ABB RobotStudio station: IRB120-Estacion.rsstn

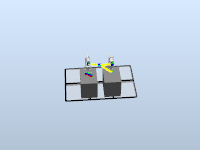
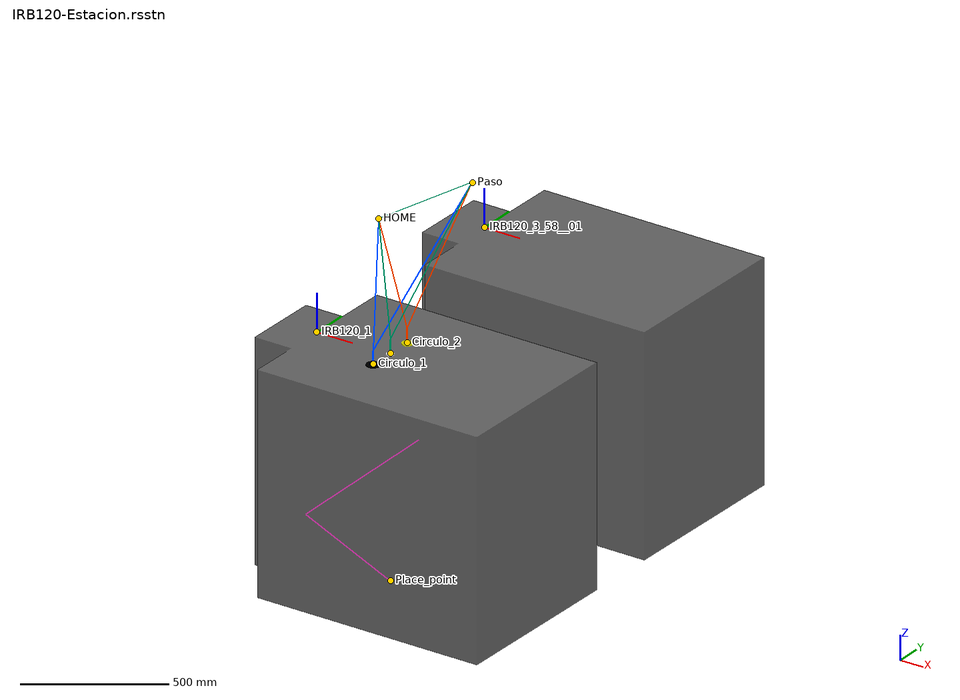
[picture v1: parts stored in the station drawn from their meshes, with robot base, taught points and paths (robot models come from the ABB library and are not in the file)]
Station IRB120 (saved by RobotStudio 21.4.9700.0)
Controller Controlador3, task T_ROB1: task frame (RAPID world) sits at (0, 980, 850) mm in the station
Controller Controlador1, task T_ROB1: task frame (RAPID world) sits at (0, 0, 850) mm in the station
Controller Controlador1
  mechanical unit ROB_1: IRB120_1, 6 joints, base frame (0, 0, 0) mm
Controller Controlador3
  mechanical unit ROB_1: IRB120_3_58__01, 6 joints, base frame (0, 0, 0) mm
Layout (positions relative to the parent item):
  - Base_2 [part] at (-150, 830, 0) mm, size 300 x 300 x 850 mm
  - IRB120_1 [mechanism, from Robots\IRB120_3_58_G_01.rslib] at (0, 0, 850) mm; joint values [0.0979, -0.2482, 0.2787, 0.0002, 1.5414, 0.0978] (rad or m)
  - Base_1 [part] at (-150, -150, 0) mm, size 300 x 300 x 850 mm
  - Ventosa_1 [mechanism, from Libraries\Ventosa.rslib] at (236.44, 23.25, 1390.49) mm, rotated rx 180 ry -0.06 rz -179.99 deg
  - Ventosa_2 [mechanism, from Libraries\Ventosa.rslib] at (364.35, 980, 1444) mm, rotated rx 180 ry 60 rz 180 deg
  - Mesa_1 [part], size 900 x 700 x 850 mm
  - Mesa_2 [part], size 900 x 700 x 850 mm
  - Circulo1 [part] at (300, 0, 850) mm, rotated rx 180 ry 0 rz 180 deg, size 30 x 29.8 x 5 mm
  - Circulo2 [part] at (300, 100, 850) mm, rotated rx 180 ry 0 rz 180 deg, size 40 x 39.8 x 5 mm
  - Circulo3 [part] at (300, -100, 850) mm, rotated rx 180 ry 0 rz 180 deg, size 50 x 49.7 x 5 mm
  - IRB120_3_58__01 [mechanism, from Robots\IRB120_3_58_G_01.rslib] at (0, 980, 850) mm; joint values [0, 0, 0, 0, 0.5236, 0] (rad or m)
Attachment: Ventosa_1 is attached to IRB120_1 / Link6
Attachment: Ventosa_2 is attached to IRB120_3_58__01 / Link6
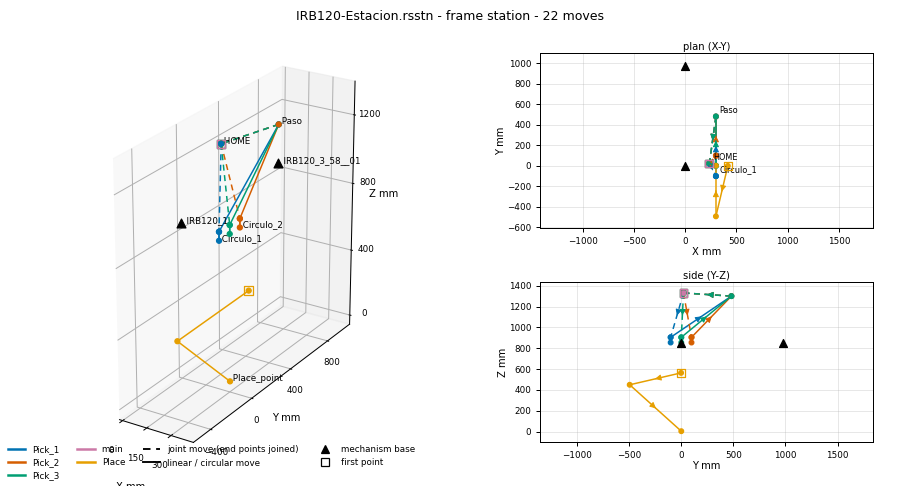
[picture p0: tool path of IRB120-Estacion.rsstn in frame station, 22 of 32 moves have a stored position in this frame; points joined in program order, loops and branches not executed]
Targets, tools, work objects and paths stored in the station, written as RAPID:
! task (no controller)
MODULE ROB1_Sim
  CONST robtarget Prueba:=[[0,0,5],[0,0,1,0],[0,0,0,0],[9E+09,9E+09,9E+09,9E+09,9E+09,9E+09]];
ENDMODULE

! task T_ROB1
MODULE ROB1_Sim
  PERS tooldata Ventosa:=[TRUE,[[0,0,60],[1,0,0,0]],[0.4,[0,0,1],[1,0,0,0],0,0,0]];
  CONST robtarget HOME:=[[236.38,23.25,480.49],[0.000528585,0.000071894,-1,-0.000034913],[0,0,0,0],[9E+09,9E+09,9E+09,9E+09,9E+09,9E+09]];
  CONST robtarget Circulo_1:=[[300,-100,5],[0,0,1,0],[-1,0,-1,0],[9E+09,9E+09,9E+09,9E+09,9E+09,9E+09]];
  CONST robtarget Circulo_2:=[[300,100,5],[0,0,1,0],[0,0,0,0],[9E+09,9E+09,9E+09,9E+09,9E+09,9E+09]];
  CONST robtarget Circulo_3:=[[300,2,5],[0,0,1,0],[0,0,0,0],[9E+09,9E+09,9E+09,9E+09,9E+09,9E+09]];
  CONST robtarget Paso:=[[300,482.5,450],[0.5,-0.5,0.5,0.5],[0,1,-1,0],[9E+09,9E+09,9E+09,9E+09,9E+09,9E+09]];
  CONST robtarget Prueba_10:=[[300,0,5],[0,0,1,0],[0,0,0,0],[9E+09,9E+09,9E+09,9E+09,9E+09,9E+09]];
  PROC Pick_1()
    MoveJ HOME,v100,fine,Ventosa\WObj:=wobj0;
    MoveJ Offs(Circulo_1,0,0,50),v100,fine,Ventosa\WObj:=wobj0;
    MoveL Circulo_1,v10,fine,Ventosa\WObj:=wobj0;
    MoveJ Offs(Circulo_1,0,0,50),v10,fine,Ventosa\WObj:=wobj0;
    MoveL Paso,v100,fine,Ventosa\WObj:=wobj0;
    MoveJ HOME,v100,fine,Ventosa\WObj:=wobj0;
  ENDPROC
  PROC Pick_2()
    MoveJ HOME,v100,fine,Ventosa\WObj:=wobj0;
    MoveJ Offs(Circulo_2,0,0,50),v100,fine,Ventosa\WObj:=wobj0;
    MoveL Circulo_2,v10,fine,Ventosa\WObj:=wobj0;
    MoveJ Offs(Circulo_2,0,0,50),v10,fine,Ventosa\WObj:=wobj0;
    MoveL Paso,v100,fine,Ventosa\WObj:=wobj0;
    MoveJ HOME,v100,fine,Ventosa\WObj:=wobj0;
  ENDPROC
  PROC Pick_3()
    MoveJ HOME,v100,fine,Ventosa\WObj:=wobj0;
    MoveJ Offs(Circulo_3,0,0,50),v100,fine,Ventosa\WObj:=wobj0;
    MoveL Circulo_3,v10,fine,Ventosa\WObj:=wobj0;
    MoveJ Offs(Circulo_3,0,0,50),v10,fine,Ventosa\WObj:=wobj0;
    MoveL Paso,v100,fine,Ventosa\WObj:=wobj0;
    MoveJ HOME,v100,fine,Ventosa\WObj:=wobj0;
  ENDPROC
ENDMODULE

! task T_ROB1
MODULE ROB1_Hanoi
  PROC main()
    MoveJ HOME,fast_speed,fine,vacuum_tool\WObj:=wobj0;
    TCP_connect;
    get_initial_state;
    TCP_close;
  ENDPROC
  PROC TCP_connect()
  ENDPROC
  PROC TCP_close()
  ENDPROC
  PROC get_initial_state()
    get_number_of_pieces;
  ENDPROC
  PROC get_number_of_pieces()
  ENDPROC
ENDMODULE

! task T_ROB1
MODULE Data
  PERS tooldata vacuum_tool:=[TRUE,[[0,0,60],[1,0,0,0]],[0.4,[0,0,1],[1,0,0,0],0,0,0]];
  TASK PERS wobjdata wo_b:=[FALSE,TRUE,"",[[448.203,36.8258,60.9458],[0.999999,-0.000331686,0.000243147,0.00150912]],[[56.8092,77.6912,0],[1,0,0,0]]];
  TASK PERS wobjdata wo_a:=[FALSE,TRUE,"",[[448.203,36.8258,60.9458],[0.999999,-0.000331686,0.000243147,0.00150912]],[[-56.0707,-122.147,0],[1,0,0,0]]];
ENDMODULE

! task T_ROB1
MODULE Hanoi_solver
  PROC initialize_desired_state()
  ENDPROC
ENDMODULE

! task T_ROB1
MODULE Module1
  PROC main()
  ENDPROC
ENDMODULE

! task T_ROB1
MODULE ROB2_Sim
  CONST robtarget HOME:=[[416.3153533,0,564],[0.5,0,0.866025404,0],[0,0,0,0],[9E+09,9E+09,9E+09,9E+09,9E+09,9E+09]];
  CONST robtarget Paso:=[[300,-492.5,450],[0.5,0.5,0.5,-0.5],[-1,-2,1,0],[9E+09,9E+09,9E+09,9E+09,9E+09,9E+09]];
  CONST robtarget Place_point:=[[300,2,5],[0,0,1,0],[0,0,0,0],[9E+09,9E+09,9E+09,9E+09,9E+09,9E+09]];
  PERS tooldata Ventosa:=[TRUE,[[0,0,60],[1,0,0,0]],[0.4,[0,0,1],[1,0,0,0],0,0,0]];
  PROC Place()
    MoveL HOME,v1000,z100,Ventosa\WObj:=wobj0;
    MoveL Paso,v1000,z100,Ventosa\WObj:=wobj0;
    MoveL Place_point,v1000,z100,Ventosa\WObj:=wobj0;
  ENDPROC
ENDMODULE

! task T_ROB1
MODULE ROB2_Hanoi
  PROC main()
    MoveJ \WObj:=wobj0;
    TCP_connect;
  ENDPROC
  PROC TCP_connect()
  ENDPROC
  PROC TCP_close()
  ENDPROC
  PROC get_initial_state()
  ENDPROC
  PROC place_on_C()
    MoveJ Offs(passing_point,0,50,0)\WObj:=wobj0;
    MoveL \WObj:=wobj0;
    WaitTime 0.5;
    MoveL Offs(passing_point,0,50,0)\WObj:=wobj0;
    MoveJ \WObj:=wobj0;
    MoveJ Offs(placing_point,0,0,(piece_height*pieces_on_C)+50);
    MoveL Offs(placing_point,0,0,(piece_height*pieces_on_C));
    WaitTime 0.5;
    MoveL Offs(placing_point,0,0,(piece_height*pieces_on_C)+50);
    MoveJ \WObj:=wobj0;
  ENDPROC
  PROC pick_and_pass()
    MoveJ Offs(placing_point,0,0,(piece_height*pieces_on_C)+50);
    MoveL Offs(placing_point,0,0,(piece_height*pieces_on_C));
    WaitTime 0.5;
    MoveL Offs(placing_point,0,0,(piece_height*pieces_on_C)+50);
    MoveJ \WObj:=wobj0;
    MoveJ Offs(passing_point,0,50,0)\WObj:=wobj0;
    MoveL \WObj:=wobj0;
    WaitTime 0.5;
    WaitTime 0.5;
    MoveL Offs(passing_point,0,50,0)\WObj:=wobj0;
    MoveJ \WObj:=wobj0;
  ENDPROC
ENDMODULE

! task T_ROB1
MODULE Module1
  CONST robtarget Target_10:=[[416.3153533,0,564],[0.5,0,0.866025404,0],[0,0,0,0],[9E+09,9E+09,9E+09,9E+09,9E+09,9E+09]];
ENDMODULE

! task T_ROB1
MODULE Data
  PERS tooldata vacuum:=[TRUE,[[0,0,0],[1,0,0,0]],[1,[0,0,0.001],[1,0,0,0],0,0,0]];
  TASK PERS wobjdata wo_c:=[FALSE,TRUE,"",[[0,0,0],[1,0,0,0]],[[0,0,0],[1,0,0,0]]];
ENDMODULE

! task T_ROB1
MODULE CalibData
  PERS tooldata Ventosa:=[TRUE,[[0,0,60],[1,0,0,0]],[0.4,[0,0,1],[1,0,0,0],0,0,0]];
ENDMODULE

